	J1=    90.000 deg,	J2=   -90.000 deg
};
P[1322]{
   GP1:
	UF : 1, UT : 1,		CONFIG : 'N U T, 0, 0, 0',
	X =  2568.524  mm,	Y =  -803.961  mm,	Z =    73.664  mm,
	W =   -43.420 deg,	P =   -13.149 deg,	R =   -17.628 deg
   GP2:
	UF : 0, UT : 1,
	J1=    90.000 deg,	J2=   -90.000 deg
};
P[1323]{
   GP1:
	UF : 1, UT : 1,		CONFIG : 'N U T, 0, 0, 0',
	X =  2648.363  mm,	Y =  -840.721  mm,	Z =   -26.432  mm,
	W =   -42.608 deg,	P =     -.037 deg,	R =    -1.279 deg
   GP2:
	UF : 0, UT : 1,
	J1=    90.000 deg,	J2=   -90.000 deg
};
P[1324]{
   GP1:
	UF : 1, UT : 1,		CONFIG : 'N U T, 0, 0, 0',
	X =  2677.162  mm,	Y =  -842.961  mm,	Z =   -27.843  mm,
	W =   -42.622 deg,	P =     -.034 deg,	R =    -1.271 deg
   GP2:
	UF : 0, UT : 1,
	J1=    90.000 deg,	J2=   -90.000 deg
};
P[1325]{
   GP1:
	UF : 1, UT : 1,		CONFIG : 'N U T, 0, 0, 0',
	X =  2692.845  mm,	Y =  -848.070  mm,	Z =   -27.626  mm,
	W =   -42.602 deg,	P =     -.050 deg,	R =   -25.548 deg
   GP2:
	UF : 0, UT : 1,
	J1=    90.000 deg,	J2=   -90.000 deg
};
P[1326]{
   GP1:
	UF : 1, UT : 1,		CONFIG : 'N U T, 0, 0, 0',
	X =  2700.985  mm,	Y =  -864.581  mm,	Z =   -26.564  mm,
	W =   -42.663 deg,	P =     -.055 deg,	R =   -39.807 deg
   GP2:
	UF : 0, UT : 1,
	J1=    90.000 deg,	J2=   -90.000 deg
};
P[1327]{
   GP1:
	UF : 1, UT : 1,		CONFIG : 'N U T, 0, 0, 0',
	X =  2739.708  mm,	Y =  -860.380  mm,	Z =    49.711  mm,
	W =   -48.781 deg,	P =    -7.527 deg,	R =   -31.543 deg
   GP2:
	UF : 0, UT : 1,
	J1=    90.000 deg,	J2=   -90.000 deg
};
P[1328]{
   GP1:
	UF : 1, UT : 1,		CONFIG : 'N U T, 0, 0, 0',
	X =  2560.230  mm,	Y =  -778.942  mm,	Z =   215.732  mm,
	W =   -62.172 deg,	P =   -18.531 deg,	R =     1.886 deg
   GP2:
	UF : 0, UT : 1,
	J1=    90.000 deg,	J2=   -90.000 deg
};
P[1329]{
   GP1:
	UF : 1, UT : 1,		CONFIG : 'N U T, 0, 0, 0',
	X =  1825.736  mm,	Y =  -967.561  mm,	Z =   255.630  mm,
	W =   -55.591 deg,	P =   -20.659 deg,	R =   -15.783 deg
   GP2:
	UF : 0, UT : 1,
	J1=    90.000 deg,	J2=   -90.000 deg
};
P[1330]{
   GP1:
	UF : 1, UT : 1,		CONFIG : 'N U T, 0, 0, 0',
	X =  1591.196  mm,	Y =  -283.866  mm,	Z =   227.110  mm,
	W =    43.884 deg,	P =    -2.387 deg,	R =     2.487 deg
   GP2:
	UF : 0, UT : 1,
	J1=    90.000 deg,	J2=   -90.000 deg
};
P[1331]{
   GP1:
	UF : 1, UT : 1,		CONFIG : 'N U T, 0, 0, 0',
	X =  1591.178  mm,	Y =  -111.276  mm,	Z =    20.110  mm,
	W =    41.925 deg,	P =   -14.562 deg,	R =    15.648 deg
   GP2:
	UF : 0, UT : 1,
	J1=    90.000 deg,	J2=   -90.000 deg
};
P[1332]{
   GP1:
	UF : 1, UT : 1,		CONFIG : 'N U T, 0, 0, 0',
	X =  1597.373  mm,	Y =   -16.036  mm,	Z =   -37.263  mm,
	W =    39.236 deg,	P =   -24.033 deg,	R =    26.523 deg
   GP2:
	UF : 0, UT : 1,
	J1=    90.000 deg,	J2=   -90.000 deg
};
P[1333]{
   GP1:
	UF : 1, UT : 1,		CONFIG : 'N U T, 0, 0, 0',
	X =  1585.811  mm,	Y =   -14.794  mm,	Z =   -38.410  mm,
	W =    39.258 deg,	P =   -24.040 deg,	R =    26.510 deg
   GP2:
	UF : 0, UT : 1,
	J1=    90.000 deg,	J2=   -90.000 deg
};
P[1334]{
   GP1:
	UF : 1, UT : 1,		CONFIG : 'N U T, 0, 0, 0',
	X =  1578.711  mm,	Y =   -17.962  mm,	Z =   -41.057  mm,
	W =    43.594 deg,	P =   -12.499 deg,	R =    37.172 deg
   GP2:
	UF : 0, UT : 1,
	J1=    90.000 deg,	J2=   -90.000 deg
};
P[1335]{
   GP1:
	UF : 1, UT : 1,		CONFIG : 'N U T, 0, 0, 0',
	X =  1573.495  mm,	Y =   -25.883  mm,	Z =   -39.530  mm,
	W =    44.958 deg,	P =    -2.238 deg,	R =    47.243 deg
   GP2:
	UF : 0, UT : 1,
	J1=    90.000 deg,	J2=   -90.000 deg
};
P[1336]{
   GP1:
	UF : 1, UT : 1,		CONFIG : 'N U T, 0, 0, 0',
	X =  1544.856  mm,	Y =   -53.211  mm,	Z =   -39.944  mm,
	W =    44.958 deg,	P =    -2.234 deg,	R =    47.237 deg
   GP2:
	UF : 0, UT : 1,
	J1=    90.000 deg,	J2=   -90.000 deg
};
P[1337]{
   GP1:
	UF : 1, UT : 1,		CONFIG : 'N U T, 0, 0, 0',
	X =  1523.602  mm,	Y =   -54.037  mm,	Z =   -39.414  mm,
	W =    34.023 deg,	P =   -31.392 deg,	R =    22.799 deg
   GP2:
	UF : 0, UT : 1,
	J1=    90.000 deg,	J2=   -90.000 deg
};
P[1338]{
   GP1:
	UF : 1, UT : 1,		CONFIG : 'N U T, 0, 0, 0',
	X =  1510.889  mm,	Y =   -43.230  mm,	Z =   -39.558  mm,
	W =   -41.192 deg,	P =   -19.995 deg,	R =    73.656 deg
   GP2:
	UF : 0, UT : 1,
	J1=    90.000 deg,	J2=   -90.000 deg
};
P[1339]{
   GP1:
	UF : 1, UT : 1,		CONFIG : 'N U T, 0, 0, 0',
	X =  1505.488  mm,	Y =     8.620  mm,	Z =   -40.409  mm,
	W =   -41.204 deg,	P =   -19.968 deg,	R =    73.684 deg
   GP2:
	UF : 0, UT : 1,
	J1=    90.000 deg,	J2=   -90.000 deg
};
P[1340]{
   GP1:
	UF : 1, UT : 1,		CONFIG : 'N U T, 0, 0, 0',
	X =  1504.857  mm,	Y =    21.151  mm,	Z =   -40.856  mm,
	W =   -32.680 deg,	P =   -32.822 deg,	R =    84.373 deg
   GP2:
	UF : 0, UT : 1,
	J1=    90.000 deg,	J2=   -90.000 deg
};
P[1341]{
   GP1:
	UF : 1, UT : 1,		CONFIG : 'N U T, 0, 0, 0',
	X =  1488.187  mm,	Y =    26.174  mm,	Z =   -42.316  mm,
	W =    -8.361 deg,	P =   -44.372 deg,	R =    89.881 deg
   GP2:
	UF : 0, UT : 1,
	J1=    90.000 deg,	J2=   -90.000 deg
};
P[1342]{
   GP1:
	UF : 1, UT : 1,		CONFIG : 'N U T, 0, 0, 0',
	X =  1464.686  mm,	Y =    30.412  mm,	Z =   -42.056  mm,
	W =    -8.369 deg,	P =   -44.373 deg,	R =    89.890 deg
   GP2:
	UF : 0, UT : 1,
	J1=    90.000 deg,	J2=   -90.000 deg
};
P[1343]{
   GP1:
	UF : 1, UT : 1,		CONFIG : 'N U T, 0, 0, 0',
	X =  1227.013  mm,	Y =  -240.395  mm,	Z =   227.364  mm,
	W =    25.573 deg,	P =   -37.026 deg,	R =    45.674 deg
   GP2:
	UF : 0, UT : 1,
	J1=    90.000 deg,	J2=   -90.000 deg
};
P[1344]{
   GP1:
	UF : 1, UT : 1,		CONFIG : 'N U T, 0, 0, 0',
	X =   647.279  mm,	Y =   337.689  mm,	Z =  -107.070  mm,
	W =    52.573 deg,	P =    53.468 deg,	R =    78.422 deg
   GP2:
	UF : 0, UT : 1,
	J1=    90.000 deg,	J2=   -90.000 deg
};
P[1345]{
   GP1:
	UF : 1, UT : 1,		CONFIG : 'N U T, 0, 0, 0',
	X =  1273.803  mm,	Y =   230.099  mm,	Z =   112.543  mm,
	W =    -1.181 deg,	P =    48.937 deg,	R =      .669 deg
   GP2:
	UF : 0, UT : 1,
	J1=    90.000 deg,	J2=   -90.000 deg
};
P[1346]{
   GP1:
	UF : 1, UT : 1,		CONFIG : 'N U T, 0, 0, 0',
	X =  1720.105  mm,	Y =   480.598  mm,	Z =    18.700  mm,
	W =    -1.280 deg,	P =    45.126 deg,	R =    -9.162 deg
   GP2:
	UF : 0, UT : 1,
	J1=    90.000 deg,	J2=   -90.000 deg
};
P[1347]{
   GP1:
	UF : 1, UT : 1,		CONFIG : 'N U T, 0, 0, 0',
	X =  1685.914  mm,	Y =   493.599  mm,	Z =   -43.455  mm,
	W =    -3.146 deg,	P =    44.903 deg,	R =   -10.505 deg
   GP2:
	UF : 0, UT : 1,
	J1=    90.000 deg,	J2=   -90.000 deg
};
P[1348]{
   GP1:
	UF : 1, UT : 1,		CONFIG : 'N U T, 0, 0, 0',
	X =  1620.065  mm,	Y =    18.872  mm,	Z =   -43.513  mm,
	W =   -38.607 deg,	P =    25.135 deg,	R =   -58.570 deg
   GP2:
	UF : 0, UT : 1,
	J1=    90.000 deg,	J2=   -90.000 deg
};
P[1349]{
   GP1:
	UF : 1, UT : 1,		CONFIG : 'N U T, 0, 0, 0',
	X =  1716.229  mm,	Y =   182.625  mm,	Z =   132.677  mm,
	W =   -40.772 deg,	P =    18.032 deg,	R =   -27.154 deg
   GP2:
	UF : 0, UT : 1,
	J1=    90.000 deg,	J2=   -90.000 deg
};
P[1350]{
   GP1:
	UF : 1, UT : 1,		CONFIG : 'N U T, 0, 0, 1',
	X =  1801.103  mm,	Y =   268.058  mm,	Z =   232.529  mm,
	W =    47.117 deg,	P =    -2.052 deg,	R =   -98.166 deg
   GP2:
	UF : 0, UT : 1,
	J1=    75.000 deg,	J2=   -90.000 deg
};
P[1351]{
   GP1:
	UF : 1, UT : 1,		CONFIG : 'N U T, 0, 0, 1',
	X =  1951.397  mm,	Y =     2.544  mm,	Z =    37.986  mm,
	W =    29.524 deg,	P =   -16.700 deg,	R =  -110.691 deg
   GP2:
	UF : 1, UT : 1,
	J1=    74.999 deg,	J2=   -90.000 deg
};
P[1352]{
   GP1:
	UF : 1, UT : 1,		CONFIG : 'N U T, 0, 0, 1',
	X =  2030.301  mm,	Y =   113.457  mm,	Z =    15.343  mm,
	W =    25.461 deg,	P =   -23.024 deg,	R =   -99.749 deg
   GP2:
	UF : 1, UT : 1,
	J1=    75.000 deg,	J2=   -90.000 deg
};
P[1353]{
   GP1:
	UF : 1, UT : 1,		CONFIG : 'N U T, 0, 0, 1',
	X =  2036.770  mm,	Y =   124.431  mm,	Z =    14.497  mm,
	W =    22.341 deg,	P =   -29.710 deg,	R =  -103.127 deg
   GP2:
	UF : 1, UT : 1,
	J1=    75.000 deg,	J2=   -90.000 deg
};
P[1354]{
   GP1:
	UF : 1, UT : 1,		CONFIG : 'N U T, 0, 0, 1',
	X =  2054.576  mm,	Y =   138.827  mm,	Z =     9.013  mm,
	W =    22.800 deg,	P =   -34.432 deg,	R =  -117.365 deg
   GP2:
	UF : 1, UT : 1,
	J1=    75.000 deg,	J2=   -90.000 deg
};
P[1355]{
   GP1:
	UF : 1, UT : 1,		CONFIG : 'N U T, 0, 0, 1',
	X =  2376.429  mm,	Y =   293.794  mm,	Z =   -73.316  mm,
	W =    -5.500 deg,	P =   -40.174 deg,	R =   -72.291 deg
   GP2:
	UF : 1, UT : 1,
	J1=    75.000 deg,	J2=   -90.000 deg
};
P[1356]{
   GP1:
	UF : 1, UT : 1,		CONFIG : 'N U T, 0, 0, 1',
	X =  2391.951  mm,	Y =   307.217  mm,	Z =   -77.744  mm,
	W =     1.457 deg,	P =   -36.015 deg,	R =   -63.555 deg
   GP2:
	UF : 1, UT : 1,
	J1=    75.000 deg,	J2=   -90.000 deg
};
P[1357]{
   GP1:
	UF : 1, UT : 1,		CONFIG : 'N U T, 0, 0, 1',
	X =  2405.655  mm,	Y =   323.649  mm,	Z =   -81.204  mm,
	W =    10.596 deg,	P =   -31.144 deg,	R =   -55.850 deg
   GP2:
	UF : 1, UT : 1,
	J1=    75.000 deg,	J2=   -90.000 deg
};
P[1358]{
   GP1:
	UF : 1, UT : 1,		CONFIG : 'N U T, 0, 0, 1',
	X =  2559.173  mm,	Y =   596.177  mm,	Z =  -120.001  mm,
	W =   -17.021 deg,	P =   -28.585 deg,	R =    -8.324 deg
   GP2:
	UF : 1, UT : 1,
	J1=    75.000 deg,	J2=   -90.000 deg
};
P[1359]{
   GP1:
	UF : 1, UT : 1,		CONFIG : 'N U T, 0, 0, 1',
	X =  2563.234  mm,	Y =   607.295  mm,	Z =  -120.021  mm,
	W =    -7.983 deg,	P =   -30.108 deg,	R =    -3.947 deg
   GP2:
	UF : 1, UT : 1,
	J1=    75.000 deg,	J2=   -90.000 deg
};
P[1360]{
   GP1:
	UF : 1, UT : 1,		CONFIG : 'N U T, 0, 0, 1',
	X =  2565.326  mm,	Y =   624.907  mm,	Z =  -121.548  mm,
	W =     6.928 deg,	P =   -29.916 deg,	R =   -19.097 deg
   GP2:
	UF : 1, UT : 1,
	J1=    75.000 deg,	J2=   -90.000 deg
};
P[1361]{
   GP1:
	UF : 1, UT : 1,		CONFIG : 'N U T, 0, 0, 0',
	X =  2551.376  mm,	Y =  1056.254  mm,	Z =  -116.499  mm,
	W =     6.097 deg,	P =   -30.066 deg,	R =     2.834 deg
   GP2:
	UF : 0, UT : 1,
	J1=    74.998 deg,	J2=   -90.000 deg
};
P[1362]{
   GP1:
	UF : 1, UT : 1,		CONFIG : 'N U T, 0, 0, 1',
	X =  2448.653  mm,	Y =  1015.496  mm,	Z =    61.125  mm,
	W =     7.047 deg,	P =   -29.835 deg,	R =     3.478 deg
   GP2:
	UF : 0, UT : 1,
	J1=    75.000 deg,	J2=   -90.000 deg
};
P[1363]{
   GP1:
	UF : 1, UT : 1,		CONFIG : 'N U T, 0, 0, 0',
	X =  1486.213  mm,	Y =   786.102  mm,	Z =   551.453  mm,
	W =   -60.827 deg,	P =   -28.283 deg,	R =    48.470 deg
   GP2:
	UF : 0, UT : 1,
	J1=    75.000 deg,	J2=   -90.000 deg
};
P[1364]{
   GP1:
	UF : 1, UT : 1,		CONFIG : 'N U T, 0, 0, 0',
	X =  2234.222  mm,	Y =  1185.195  mm,	Z =   220.863  mm,
	W =    10.036 deg,	P =   -28.420 deg,	R =   -20.397 deg
   GP2:
	UF : 0, UT : 1,
	J1=    75.000 deg,	J2=   -90.000 deg
};
P[1365]{
   GP1:
	UF : 1, UT : 1,		CONFIG : 'N U T, 0, 0, 0',
	X =  2409.709  mm,	Y =  1193.069  mm,	Z =   -77.360  mm,
	W =    10.002 deg,	P =   -28.454 deg,	R =   -20.362 deg
   GP2:
	UF : 0, UT : 1,
	J1=    75.000 deg,	J2=   -90.000 deg
};
P[1366]{
   GP1:
	UF : 1, UT : 1,		CONFIG : 'N U T, 0, 0, 0',
	X =  2410.536  mm,	Y =  1173.522  mm,	Z =   -78.269  mm,
	W =    10.723 deg,	P =   -28.212 deg,	R =   -20.271 deg
   GP2:
	UF : 1, UT : 1,
	J1=    75.000 deg,	J2=   -90.000 deg
};
P[1367]{
   GP1:
	UF : 1, UT : 1,		CONFIG : 'N U T, 0, 0, 0',
	X =  2416.768  mm,	Y =  1169.024  mm,	Z =   -81.705  mm,
	W =    10.551 deg,	P =   -24.468 deg,	R =     4.981 deg
   GP2:
	UF : 0, UT : 1,
	J1=    74.999 deg,	J2=   -90.000 deg
};
P[1368]{
   GP1:
	UF : 1, UT : 1,		CONFIG : 'N U T, 0, 0, 0',
	X =  2427.010  mm,	Y =  1167.278  mm,	Z =   -87.519  mm,
	W =    39.646 deg,	P =    27.550 deg,	R =   -14.663 deg
   GP2:
	UF : 0, UT : 1,
	J1=    74.999 deg,	J2=   -90.000 deg
};
P[1369]{
   GP1:
	UF : 1, UT : 1,		CONFIG : 'N U T, 0, 0, 0',
	X =  2441.825  mm,	Y =  1166.073  mm,	Z =   -89.180  mm,
	W =    39.628 deg,	P =    27.532 deg,	R =   -14.658 deg
   GP2:
	UF : 0, UT : 1,
	J1=    75.000 deg,	J2=   -90.000 deg
};
P[1370]{
   GP1:
	UF : 1, UT : 1,		CONFIG : 'N U T, 0, 0, 0',
	X =  2470.501  mm,	Y =  1161.239  mm,	Z =   -97.706  mm,
	W =    38.840 deg,	P =    12.983 deg,	R =   -24.465 deg
   GP2:
	UF : 0, UT : 1,
	J1=    75.000 deg,	J2=   -90.000 deg
};
P[1371]{
   GP1:
	UF : 1, UT : 1,		CONFIG : 'N U T, 0, 0, 0',
	X =  2500.305  mm,	Y =  1139.803  mm,	Z =  -105.226  mm,
	W =    35.674 deg,	P =     -.854 deg,	R =   -29.753 deg
   GP2:
	UF : 0, UT : 1,
	J1=    75.000 deg,	J2=   -90.000 deg
};
P[1372]{
   GP1:
	UF : 1, UT : 1,		CONFIG : 'N U T, 0, 0, 0',
	X =  2536.842  mm,	Y =  1100.347  mm,	Z =  -115.023  mm,
	W =    35.543 deg,	P =    -1.138 deg,	R =   -29.936 deg
   GP2:
	UF : 0, UT : 1,
	J1=    75.000 deg,	J2=   -90.000 deg
};
P[1373]{
   GP1:
	UF : 1, UT : 1,		CONFIG : 'N U T, 0, 0, 0',
	X =  2546.545  mm,	Y =  1081.318  mm,	Z =  -117.080  mm,
	W =    25.189 deg,	P =   -20.016 deg,	R =   -20.921 deg
   GP2:
	UF : 0, UT : 1,
	J1=    75.000 deg,	J2=   -90.000 deg
};
P[1374]{
   GP1:
	UF : 1, UT : 1,		CONFIG : 'N U T, 0, 0, 0',
	X =  2550.840  mm,	Y =  1055.699  mm,	Z =  -118.307  mm,
	W =    19.755 deg,	P =   -23.078 deg,	R =   -38.813 deg
   GP2:
	UF : 0, UT : 1,
	J1=    75.000 deg,	J2=   -90.000 deg
};
P[1375]{
   GP1:
	UF : 1, UT : 1,		CONFIG : 'N U T, 0, 0, 0',
	X =  2429.591  mm,	Y =   941.223  mm,	Z =   111.356  mm,
	W =    40.532 deg,	P =   -18.229 deg,	R =   -35.810 deg
   GP2:
	UF : 0, UT : 1,
	J1=    75.000 deg,	J2=   -90.000 deg
};
P[1376]{
   GP1:
	UF : 1, UT : 1,		CONFIG : 'N U T, 0, 0, 0',
	X =  1135.590  mm,	Y =   941.223  mm,	Z =   631.357  mm,
	W =    40.532 deg,	P =   -18.229 deg,	R =   -35.810 deg
   GP2:
	UF : 0, UT : 1,
	J1=    75.000 deg,	J2=   -90.000 deg
};
P[1377]{
   GP1:
	UF : 1, UT : 1,		CONFIG : 'N U T, 0, 0, -1',
	X =   594.691  mm,	Y =   765.878  mm,	Z =  1492.090  mm,
	W =   -20.214 deg,	P =    51.430 deg,	R =  -175.387 deg
   GP2:
	UF : 0, UT : 1,
	J1=    75.000 deg,	J2=   -90.000 deg
};
P[1378]{
   GP1:
	UF : 1, UT : 1,		CONFIG : 'N U T, 0, 0, 0',
	X =   897.328  mm,	Y =   -44.116  mm,	Z =  1758.586  mm,
	W =    -8.576 deg,	P =    70.752 deg,	R =  -170.008 deg
   GP2:
	UF : 0, UT : 1,
	J1=    75.000 deg,	J2=   -90.000 deg
};
P[1379]{
   GP1:
	UF : 1, UT : 1,		CONFIG : 'N U T, 0, 0, 0',
	X =  2053.676  mm,	Y =  -119.321  mm,	Z =  1258.210  mm,
	W =    -3.043 deg,	P =    35.787 deg,	R =  -167.926 deg
   GP2:
	UF : 0, UT : 1,
	J1=    90.000 deg,	J2=   -90.000 deg
};
P[1380]{
   GP1:
	UF : 1, UT : 1,		CONFIG : 'N U T, 0, 0, 0',
	X =  2059.608  mm,	Y =  -129.321  mm,	Z =   981.210  mm,
	W =    -3.043 deg,	P =    35.787 deg,	R =  -167.926 deg
   GP2:
	UF : 0, UT : 1,
	J1=    90.000 deg,	J2=   -90.000 deg
};
P[1381]{
   GP1:
	UF : 1, UT : 1,		CONFIG : 'N U T, 0, 0, 0',
	X =  2081.803  mm,	Y =  -104.576  mm,	Z =   863.928  mm,
	W =    -4.711 deg,	P =    44.807 deg,	R =  -168.724 deg
   GP2:
	UF : 0, UT : 1,
	J1=    90.000 deg,	J2=   -90.000 deg
};
P[1382]{
   GP1:
	UF : 1, UT : 1,		CONFIG : 'N U T, 0, 0, 0',
	X =  2076.243  mm,	Y =   -76.244  mm,	Z =   862.598  mm,
	W =    -4.760 deg,	P =    44.804 deg,	R =  -168.727 deg
   GP2:
	UF : 0, UT : 1,
	J1=    89.999 deg,	J2=   -90.000 deg
};
P[1383]{
   GP1:
	UF : 1, UT : 1,		CONFIG : 'N U T, 0, 0, 0',
	X =  2060.180  mm,	Y =   -62.212  mm,	Z =   862.114  mm,
	W =    -5.900 deg,	P =    44.717 deg,	R =   -77.457 deg
   GP2:
	UF : 0, UT : 1,
	J1=    89.999 deg,	J2=   -90.000 deg
};
P[1384]{
   GP1:
	UF : 1, UT : 1,		CONFIG : 'N U T, 0, 0, 0',
	X =  2033.586  mm,	Y =   -85.112  mm,	Z =   859.812  mm,
	W =    -1.775 deg,	P =    44.967 deg,	R =    10.202 deg
   GP2:
	UF : 0, UT : 1,
	J1=    90.000 deg,	J2=   -90.000 deg
};
P[1385]{
   GP1:
	UF : 1, UT : 1,		CONFIG : 'N U T, 0, 0, 0',
	X =  2042.594  mm,	Y =  -111.090  mm,	Z =   859.808  mm,
	W =    -5.461 deg,	P =    44.730 deg,	R =    10.235 deg
   GP2:
	UF : 0, UT : 1,
	J1=    90.000 deg,	J2=   -90.000 deg
};
P[1386]{
   GP1:
	UF : 1, UT : 1,		CONFIG : 'N U T, 0, 0, 0',
	X =  2072.668  mm,	Y =  -118.651  mm,	Z =   860.814  mm,
	W =    -1.333 deg,	P =    44.974 deg,	R =   112.384 deg
   GP2:
	UF : 0, UT : 1,
	J1=    90.000 deg,	J2=   -90.000 deg
};
P[1387]{
   GP1:
	UF : 1, UT : 1,		CONFIG : 'N U T, 0, 0, 1',
	X =  2084.006  mm,	Y =  -100.733  mm,	Z =   863.362  mm,
	W =      .144 deg,	P =    45.003 deg,	R =  -161.772 deg
   GP2:
	UF : 0, UT : 1,
	J1=    90.000 deg,	J2=   -90.000 deg
};
P[1388]{
   GP1:
	UF : 1, UT : 1,		CONFIG : 'N U T, 0, 0, 1',
	X =  2044.049  mm,	Y =  -114.041  mm,	Z =  1004.475  mm,
	W =      .165 deg,	P =    45.000 deg,	R =  -161.765 deg
   GP2:
	UF : 0, UT : 1,
	J1=    90.000 deg,	J2=   -90.000 deg
};
P[1389]{
   GP1:
	UF : 1, UT : 1,		CONFIG : 'N U T, 0, 0, 0',
	X =  2081.406  mm,	Y =  -215.644  mm,	Z =  1032.770  mm,
	W =    -3.996 deg,	P =    46.100 deg,	R =   -98.107 deg
   GP2:
	UF : 0, UT : 1,
	J1=    90.000 deg,	J2=   -90.000 deg
};
P[1390]{
   GP1:
	UF : 1, UT : 1,		CONFIG : 'N U T, 0, 0, 0',
	X =  2057.931  mm,	Y =  -158.349  mm,	Z =   860.063  mm,
	W =    -5.604 deg,	P =    44.746 deg,	R =   -97.938 deg
   GP2:
	UF : 0, UT : 1,
	J1=    90.000 deg,	J2=   -90.000 deg
};
P[1391]{
   GP1:
	UF : 1, UT : 1,		CONFIG : 'N U T, 0, 0, 0',
	X =  2181.282  mm,	Y =  -156.646  mm,	Z =   861.080  mm,
	W =    -5.610 deg,	P =    44.738 deg,	R =   -97.948 deg
   GP2:
	UF : 0, UT : 1,
	J1=    90.000 deg,	J2=   -90.000 deg
};
P[1392]{
   GP1:
	UF : 1, UT : 1,		CONFIG : 'N U T, 0, 0, 0',
	X =  2222.260  mm,	Y =  -138.497  mm,	Z =   861.141  mm,
	W =    -8.257 deg,	P =    44.429 deg,	R =   -63.806 deg
   GP2:
	UF : 0, UT : 1,
	J1=    89.999 deg,	J2=   -90.000 deg
};
P[1393]{
   GP1:
	UF : 1, UT : 1,		CONFIG : 'N U T, 0, 0, 0',
	X =  2247.668  mm,	Y =   -98.898  mm,	Z =   862.440  mm,
	W =    -6.114 deg,	P =    44.679 deg,	R =   -22.818 deg
   GP2:
	UF : 0, UT : 1,
	J1=    90.000 deg,	J2=   -90.000 deg
};
P[1394]{
   GP1:
	UF : 1, UT : 1,		CONFIG : 'N U T, 0, 0, 0',
	X =  2355.337  mm,	Y =    57.690  mm,	Z =   866.973  mm,
	W =    20.402 deg,	P =    41.026 deg,	R =   -23.468 deg
   GP2:
	UF : 0, UT : 1,
	J1=    90.000 deg,	J2=   -90.000 deg
};
P[1395]{
   GP1:
	UF : 1, UT : 1,		CONFIG : 'N U T, 0, 0, 0',
	X =  2547.015  mm,	Y =    98.417  mm,	Z =   868.417  mm,
	W =    39.275 deg,	P =    24.127 deg,	R =   -34.882 deg
   GP2:
	UF : 0, UT : 1,
	J1=    89.999 deg,	J2=   -90.000 deg
};
P[1396]{
   GP1:
	UF : 1, UT : 1,		CONFIG : 'N U T, 0, 0, 0',
	X =  2598.256  mm,	Y =   116.207  mm,	Z =   863.365  mm,
	W =    11.867 deg,	P =    45.051 deg,	R =   -52.690 deg
   GP2:
	UF : 0, UT : 1,
	J1=    89.999 deg,	J2=   -90.000 deg
};
P[1397]{
   GP1:
	UF : 1, UT : 1,		CONFIG : 'N U T, 0, 0, 0',
	X =  2626.706  mm,	Y =   158.484  mm,	Z =   864.421  mm,
	W =    26.734 deg,	P =    37.663 deg,	R =    -3.650 deg
   GP2:
	UF : 0, UT : 1,
	J1=    89.999 deg,	J2=   -90.000 deg
};
P[1398]{
   GP1:
	UF : 1, UT : 1,		CONFIG : 'N U T, 0, 0, 0',
	X =  2666.149  mm,	Y =   165.388  mm,	Z =  1006.200  mm,
	W =    23.231 deg,	P =    35.687 deg,	R =   -21.225 deg
   GP2:
	UF : 0, UT : 1,
	J1=    90.000 deg,	J2=   -90.000 deg
};
P[1399]{
   GP1:
	UF : 1, UT : 1,		CONFIG : 'N U T, 0, 0, 0',
	X =  2360.151  mm,	Y =    86.388  mm,	Z =   981.215  mm,
	W =    23.231 deg,	P =    35.687 deg,	R =   -21.225 deg
   GP2:
	UF : 0, UT : 1,
	J1=    90.000 deg,	J2=   -90.000 deg
};
P[1400]{
   GP1:
	UF : 1, UT : 1,		CONFIG : 'N U T, 0, 0, 0',
	X =  2350.101  mm,	Y =   138.579  mm,	Z =   874.539  mm,
	W =    23.286 deg,	P =    35.713 deg,	R =   -27.094 deg
   GP2:
	UF : 0, UT : 1,
	J1=    89.999 deg,	J2=   -90.000 deg
};
P[1401]{
   GP1:
	UF : 1, UT : 1,		CONFIG : 'N U T, 0, 0, 0',
	X =  2284.041  mm,	Y =   104.828  mm,	Z =   873.193  mm,
	W =    23.235 deg,	P =    35.686 deg,	R =   -27.115 deg
   GP2:
	UF : 0, UT : 1,
	J1=    90.000 deg,	J2=   -90.000 deg
};
P[1402]{
   GP1:
	UF : 1, UT : 1,		CONFIG : 'N U T, 0, 0, 0',
	X =  2318.792  mm,	Y =    59.786  mm,	Z =   930.546  mm,
	W =    22.474 deg,	P =    36.128 deg,	R =   -18.977 deg
   GP2:
	UF : 0, UT : 1,
	J1=    90.000 deg,	J2=   -90.000 deg
};
P[1403]{
   GP1:
	UF : 1, UT : 1,		CONFIG : 'N U T, 0, 0, 0',
	X =  2383.594  mm,	Y =   190.187  mm,	Z =   944.949  mm,
	W =     2.802 deg,	P =    41.645 deg,	R =    35.577 deg
   GP2:
	UF : 0, UT : 1,
	J1=    90.000 deg,	J2=   -90.000 deg
};
P[1404]{
   GP1:
	UF : 1, UT : 1,		CONFIG : 'N U T, 0, 0, 0',
	X =  2338.561  mm,	Y =   165.143  mm,	Z =   872.108  mm,
	W =     2.819 deg,	P =    41.634 deg,	R =    35.579 deg
   GP2:
	UF : 0, UT : 1,
	J1=    90.000 deg,	J2=   -90.000 deg
};
P[1405]{
   GP1:
	UF : 1, UT : 1,		CONFIG : 'N U T, 0, 0, 0',
	X =  2350.265  mm,	Y =   140.419  mm,	Z =   871.898  mm,
	W =     2.806 deg,	P =    41.648 deg,	R =    35.590 deg
   GP2:
	UF : 0, UT : 1,
	J1=    90.000 deg,	J2=   -90.000 deg
};
P[1406]{
   GP1:
	UF : 1, UT : 1,		CONFIG : 'N U T, 0, 0, 0',
	X =  2394.447  mm,	Y =   159.675  mm,	Z =   934.277  mm,
	W =     2.802 deg,	P =    41.645 deg,	R =    35.577 deg
   GP2:
	UF : 0, UT : 1,
	J1=    90.000 deg,	J2=   -90.000 deg
};
P[1407]{
   GP1:
	UF : 1, UT : 1,		CONFIG : 'N U T, 0, 0, 0',
	X =  2237.352  mm,	Y =   151.375  mm,	Z =   981.847  mm,
	W =   -31.407 deg,	P =    29.635 deg,	R =    66.585 deg
   GP2:
	UF : 0, UT : 1,
	J1=    90.000 deg,	J2=   -90.000 deg
};
P[1408]{
   GP1:
	UF : 1, UT : 1,		CONFIG : 'N U T, 0, 0, 0',
	X =  2268.643  mm,	Y =   130.272  mm,	Z =   874.453  mm,
	W =   -30.491 deg,	P =    30.803 deg,	R =    76.658 deg
   GP2:
	UF : 0, UT : 1,
	J1=    90.000 deg,	J2=   -90.000 deg
};
P[1409]{
   GP1:
	UF : 1, UT : 1,		CONFIG : 'N U T, 0, 0, 0',
	X =  2334.675  mm,	Y =   163.679  mm,	Z =   874.552  mm,
	W =   -30.712 deg,	P =    31.401 deg,	R =    76.553 deg
   GP2:
	UF : 0, UT : 1,
	J1=    90.000 deg,	J2=   -90.000 deg
};
P[1410]{
   GP1:
	UF : 1, UT : 1,		CONFIG : 'N U T, 0, 0, 0',
	X =  2301.976  mm,	Y =   199.747  mm,	Z =   934.083  mm,
	W =   -30.368 deg,	P =    30.111 deg,	R =    93.411 deg
   GP2:
	UF : 0, UT : 1,
	J1=    90.000 deg,	J2=   -90.000 deg
};
P[1411]{
   GP1:
	UF : 1, UT : 1,		CONFIG : 'N U T, 0, 0, 0',
	X =  1939.340  mm,	Y =   134.263  mm,	Z =   990.229  mm,
	W =   -27.894 deg,	P =    40.770 deg,	R =   134.668 deg
   GP2:
	UF : 0, UT : 1,
	J1=    90.000 deg,	J2=   -90.000 deg
};
P[1412]{
   GP1:
	UF : 1, UT : 1,		CONFIG : 'N U T, 0, 0, 0',
	X =  1538.072  mm,	Y =    68.062  mm,	Z =   943.499  mm,
	W =   -27.896 deg,	P =    40.772 deg,	R =   140.108 deg
   GP2:
	UF : 0, UT : 1,
	J1=    90.000 deg,	J2=   -90.000 deg
};
P[1413]{
   GP1:
	UF : 1, UT : 1,		CONFIG : 'N U T, 0, 0, 0',
	X =  1598.420  mm,	Y =    65.212  mm,	Z =   867.697  mm,
	W =   -27.906 deg,	P =    40.774 deg,	R =   140.097 deg
   GP2:
	UF : 0, UT : 1,
	J1=    89.999 deg,	J2=   -90.000 deg
};
P[1414]{
   GP1:
	UF : 1, UT : 1,		CONFIG : 'N U T, 0, 0, 0',
	X =  1669.618  mm,	Y =   567.250  mm,	Z =   869.620  mm,
	W =   -42.379 deg,	P =    24.896 deg,	R =   114.371 deg
   GP2:
	UF : 0, UT : 1,
	J1=    89.994 deg,	J2=   -90.001 deg
};
P[1415]{
   GP1:
	UF : 1, UT : 1,		CONFIG : 'N U T, 0, 0, 0',
	X =  1660.119  mm,	Y =   593.490  mm,	Z =   950.317  mm,
	W =   -47.316 deg,	P =    14.922 deg,	R =   119.101 deg
   GP2:
	UF : 0, UT : 1,
	J1=    90.000 deg,	J2=   -90.000 deg
};
P[1416]{
   GP1:
	UF : 1, UT : 1,		CONFIG : 'N U T, 0, 0, 0',
	X =  1684.004  mm,	Y =   511.820  mm,	Z =   999.263  mm,
	W =   -44.984 deg,	P =    18.872 deg,	R =   121.131 deg
   GP2:
	UF : 0, UT : 1,
	J1=    89.999 deg,	J2=   -90.000 deg
};
P[1417]{
   GP1:
	UF : 1, UT : 1,		CONFIG : 'N U T, 0, 0, 0',
	X =  1749.421  mm,	Y =   289.455  mm,	Z =   974.394  mm,
	W =    -1.202 deg,	P =     4.318 deg,	R =    75.209 deg
   GP2:
	UF : 0, UT : 1,
	J1=    89.999 deg,	J2=   -90.000 deg
};
P[1418]{
   GP1:
	UF : 1, UT : 1,		CONFIG : 'N U T, 0, 0, 0',
	X =  1695.312  mm,	Y =    49.332  mm,	Z =   945.661  mm,
	W =    36.232 deg,	P =    29.646 deg,	R =    39.019 deg
   GP2:
	UF : 0, UT : 1,
	J1=    89.999 deg,	J2=   -90.000 deg
};
P[1419]{
   GP1:
	UF : 1, UT : 1,		CONFIG : 'N U T, 0, 0, 0',
	X =  1622.505  mm,	Y =    65.119  mm,	Z =   870.110  mm,
	W =    36.239 deg,	P =    29.632 deg,	R =    39.026 deg
   GP2:
	UF : 0, UT : 1,
	J1=    89.998 deg,	J2=   -90.000 deg
};
P[1420]{
   GP1:
	UF : 1, UT : 1,		CONFIG : 'N U T, 0, 0, 0',
	X =  1689.469  mm,	Y =   572.225  mm,	Z =   869.908  mm,
	W =    40.571 deg,	P =    22.639 deg,	R =    50.196 deg
   GP2:
	UF : 0, UT : 1,
	J1=    89.999 deg,	J2=   -90.000 deg
};
P[1421]{
   GP1:
	UF : 1, UT : 1,		CONFIG : 'N U T, 0, 0, 0',
	X =  1772.810  mm,	Y =   561.424  mm,	Z =   953.851  mm,
	W =    39.352 deg,	P =    13.418 deg,	R =    41.887 deg
   GP2:
	UF : 0, UT : 1,
	J1=    89.999 deg,	J2=   -90.000 deg
};
P[1422]{
   GP1:
	UF : 1, UT : 1,		CONFIG : 'N U T, 0, 0, 0',
	X =  1146.298  mm,	Y = -1473.938  mm,	Z =  1607.148  mm,
	W =   -45.551 deg,	P =   -20.029 deg,	R =   -44.051 deg
   GP2:
	UF : 0, UT : 1,
	J1=    90.000 deg,	J2=   -80.000 deg
};
P[1423]{
   GP1:
	UF : 1, UT : 1,		CONFIG : 'F U T, 0, 0, 0',
	X =  2545.462  mm,	Y = -1553.476  mm,	Z =  1146.714  mm,
	W =   -35.769 deg,	P =   -28.014 deg,	R =    20.274 deg
   GP2:
	UF : 0, UT : 1,
	J1=    90.000 deg,	J2=   -80.000 deg
};
P[1424]{
   GP1:
	UF : 1, UT : 1,		CONFIG : 'F U T, 0, 0, 0',
	X =  2486.860  mm,	Y = -1628.009  mm,	Z =   967.791  mm,
	W =   -35.088 deg,	P =   -31.677 deg,	R =    63.073 deg
   GP2:
	UF : 0, UT : 1,
	J1=    90.000 deg,	J2=   -80.000 deg
};
P[1425]{
   GP1:
	UF : 1, UT : 1,		CONFIG : 'F U T, 0, 0, 0',
	X =  2755.354  mm,	Y = -1563.841  mm,	Z =   703.375  mm,
	W =   -35.088 deg,	P =   -31.677 deg,	R =    63.073 deg
   GP2:
	UF : 0, UT : 1,
	J1=    90.000 deg,	J2=   -80.000 deg
};
P[1426]{
   GP1:
	UF : 1, UT : 1,		CONFIG : 'F U T, 0, 0, 0',
	X =  2860.518  mm,	Y = -1474.004  mm,	Z =   619.430  mm,
	W =   -11.515 deg,	P =   -49.293 deg,	R =    46.708 deg
   GP2:
	UF : 1, UT : 1,
	J1=    89.999 deg,	J2=   -80.000 deg
};
P[1427]{
   GP1:
	UF : 1, UT : 1,		CONFIG : 'F U T, 0, 0, 0',
	X =  2861.805  mm,	Y = -1511.751  mm,	Z =   614.512  mm,
	W =   -37.671 deg,	P =   -31.187 deg,	R =    57.797 deg
   GP2:
	UF : 1, UT : 1,
	J1=    89.999 deg,	J2=   -80.000 deg
};
P[1428]{
   GP1:
	UF : 1, UT : 1,		CONFIG : 'F U T, 0, 0, 0',
	X =  2846.945  mm,	Y = -1554.557  mm,	Z =   608.687  mm,
	W =   -41.709 deg,	P =   -23.013 deg,	R =    48.917 deg
   GP2:
	UF : 1, UT : 1,
	J1=    89.999 deg,	J2=   -80.000 deg
};
P[1429]{
   GP1:
	UF : 1, UT : 1,		CONFIG : 'F U T, 0, 0, 0',
	X =  2817.070  mm,	Y = -1584.013  mm,	Z =   601.641  mm,
	W =   -37.085 deg,	P =   -21.237 deg,	R =    24.447 deg
   GP2:
	UF : 1, UT : 1,
	J1=    89.999 deg,	J2=   -80.000 deg
};
P[1430]{
   GP1:
	UF : 1, UT : 1,		CONFIG : 'F U T, 0, 0, 0',
	X =  2760.403  mm,	Y = -1616.161  mm,	Z =   596.052  mm,
	W =   -37.129 deg,	P =   -21.189 deg,	R =    22.320 deg
   GP2:
	UF : 1, UT : 1,
	J1=    89.999 deg,	J2=   -80.000 deg
};
P[1431]{
   GP1:
	UF : 1, UT : 1,		CONFIG : 'F U T, 0, 0, 0',
	X =  2701.350  mm,	Y = -1572.365  mm,	Z =   665.669  mm,
	W =   -43.039 deg,	P =   -10.740 deg,	R =    31.361 deg
   GP2:
	UF : 0, UT : 1,
	J1=    90.000 deg,	J2=   -80.000 deg
};
P[1432]{
   GP1:
	UF : 1, UT : 1,		CONFIG : 'F U T, 0, 0, 0',
	X =  2604.020  mm,	Y = -1663.100  mm,	Z =   852.581  mm,
	W =  -106.889 deg,	P =    58.736 deg,	R =    44.006 deg
   GP2:
	UF : 0, UT : 1,
	J1=    90.000 deg,	J2=   -80.000 deg
};
P[1433]{
   GP1:
	UF : 1, UT : 1,		CONFIG : 'F U T, 0, 0, 0',
	X =  2652.666  mm,	Y = -1671.679  mm,	Z =   674.601  mm,
	W =    47.958 deg,	P =    12.926 deg,	R =   -63.288 deg
   GP2:
	UF : 0, UT : 1,
	J1=    90.000 deg,	J2=   -80.000 deg
};
P[1434]{
   GP1:
	UF : 1, UT : 1,		CONFIG : 'F U T, 0, 0, 0',
	X =  2762.218  mm,	Y = -1619.799  mm,	Z =   593.853  mm,
	W =    49.059 deg,	P =    13.941 deg,	R =   -64.255 deg
   GP2:
	UF : 1, UT : 1,
	J1=    89.999 deg,	J2=   -80.000 deg
};
P[1435]{
   GP1:
	UF : 1, UT : 1,		CONFIG : 'F U T, 0, 0, 0',
	X =  2778.298  mm,	Y = -1646.308  mm,	Z =   589.867  mm,
	W =    49.121 deg,	P =    13.967 deg,	R =   -64.229 deg
   GP2:
	UF : 1, UT : 1,
	J1=    89.999 deg,	J2=   -80.000 deg
};
P[1436]{
   GP1:
	UF : 1, UT : 1,		CONFIG : 'F U T, 0, 0, 0',
	X =  2710.694  mm,	Y = -1669.180  mm,	Z =   631.558  mm,
	W =    48.076 deg,	P =     9.473 deg,	R =   -69.425 deg
   GP2:
	UF : 0, UT : 1,
	J1=    90.000 deg,	J2=   -80.000 deg
};
P[1437]{
   GP1:
	UF : 1, UT : 1,		CONFIG : 'F U T, 0, 0, 0',
	X =  2442.025  mm,	Y = -1810.445  mm,	Z =  1068.442  mm,
	W =    50.396 deg,	P =     5.479 deg,	R =   -69.123 deg
   GP2:
	UF : 0, UT : 1,
	J1=    90.000 deg,	J2=   -80.000 deg
};
P[1438]{
   GP1:
	UF : 1, UT : 1,		CONFIG : 'F U T, 0, 0, 0',
	X =  1897.508  mm,	Y = -1522.490  mm,	Z =  2080.903  mm,
	W =    58.754 deg,	P =   -40.157 deg,	R =   -73.858 deg
   GP2:
	UF : 0, UT : 1,
	J1=    90.000 deg,	J2=   -80.000 deg
};
/END
